# EPICS substitutions: op-vlspgm/PGM/db/PGM_IOCsystem.substitutions
# DEVICE: device name
# CARD:
# CS_VERSION_VAL

file /epics/pgm/modules/uIOCSystem/db/system.template {
pattern { DEVICE, CARD, CS_VERSION_VAL}
	{ "FMBPGMIOC01", "0", "testing" }
}

#EOF
